{attribute 'linkalways'} 
{attribute 'no_explicit_call' := 'This FB is a CLASS and must be accessed using methods or properties'}
{attribute 'enable_dynamic_creation'}
FUNCTION_BLOCK _ETcVnRTrees EXTENDS EnumDatatypeBase
VAR
	localData : ETcVnRTrees;
	activeData : REFERENCE TO ETcVnRTrees;
	enumBaseDatatype : _UDINT(localData);
END_VAR

METHOD PRIVATE AddLocalEnumeration
VAR_INPUT
	Enumeration : T_MAXSTRING;
	Value : ETcVnRTrees;
END_VAR
AddEnumeration(Enumeration, Value);
END_METHOD

PROPERTY PUBLIC Address : PVOID
GET
Address := ADR(activeData);
END_GET
END_PROPERTY

METHOD PUBLIC ClearReference
VAR_INPUT
END_VAR
activeData REF= localData;
SetBaseDatatypeReference();
END_METHOD

METHOD PUBLIC Clone : I_Datatype
VAR
    pClone : POINTER TO _ETcVnRTrees;
END_VAR
pClone := __NEW(_ETcVnRTrees(InitialValue := Value));
Clone := pClone^;
END_METHOD

METHOD FB_init : BOOL
VAR_INPUT
	bInitRetains : BOOL; // if TRUE, the retain variables are initialized (warm start / cold start)
	bInCopyCode : BOOL;  // if TRUE, the instance afterwards gets moved into the copy code (online change)
	InitialValue : ETcVnRTrees;
END_VAR
localData := InitialValue;
AddBaseDatatype(enumBaseDatatype);
ClearReference();

AddLocalEnumeration('TCVN_RT_CLASSIFIER', ETcVnRTrees.TCVN_RT_CLASSIFIER);
AddLocalEnumeration('TCVN_RT_REGRESSOR', ETcVnRTrees.TCVN_RT_REGRESSOR);
END_METHOD

PROPERTY PUBLIC Identifier : T_MAXSTRING
GET
Identifier := 'ETcVnRTrees';
END_GET
END_PROPERTY

METHOD IsEnumeratorValueEqual : BOOL
VAR_INPUT
	Enumerator : I_KeyValueForwardEnumerator;
END_VAR
VAR
	storedValue : ETcVnRTrees;
END_VAR
IF NOT Enumerator.TryGet(storedValue) THEN
	RETURN;
END_IF

IsEnumeratorValueEqual := storedValue = activeData;
END_METHOD

METHOD PUBLIC MakeReferenceTo
VAR_INPUT
	ReferenceTarget : REFERENCE TO ETcVnRTrees;
END_VAR
activeData REF= ReferenceTarget;
SetBaseDatatypeReference();
END_METHOD

METHOD PROTECTED SetBaseDatatypeReference
VAR_INPUT
END_VAR
enumBaseDatatype.MakeReferenceTo(activeData);
END_METHOD

PROPERTY PUBLIC Size : UDINT
GET
Size := SIZEOF(activeData);
END_GET
END_PROPERTY

METHOD TryMakeReferenceTo : BOOL
VAR_INPUT
	Target : I_Datatype;
END_VAR
VAR
	targetAsEnum : I_EnumDatatype;
	pTargetData : POINTER TO ETcVnRTrees;
END_VAR
IF NOT Target.TryResolveAsEnumDatatype(targetAsEnum) THEN
	RETURN;
END_IF

IF targetAsEnum.Identifier <> Identifier THEN
	RETURN;
END_IF

pTargetData := Target.Address;
activeData REF= pTargetData^;
SetBaseDatatypeReference();
TryMakeReferenceTo := TRUE;
END_METHOD

PROPERTY PUBLIC Value : ETcVnRTrees
GET
Value := activeData;
END_GET
SET
activeData := Value;
END_SET
END_PROPERTY

END_FUNCTION_BLOCK

(* stored: Version 1.1.0.1, ProductVersion 3.1.4024.12
   POU _ETcVnRTrees: Id {5121f43b-3ca2-4baf-bd5c-a2722b22dd51}, SpecialFunc None
   Folder Constructor: Id {2dcca765-5c1c-4e5d-8a56-08c78f1e00a4}
   Folder Private: Id {82459e84-156f-4780-8edb-40ba5a89ab1f}
   Folder Protected: Id {f1614cfd-2cbd-46a2-8779-fde5d5b4e889}
   Method AddLocalEnumeration: Id {f0e52ad1-1d34-4ede-a2cc-4e0a7a0d8418}
   Property Address: Id {9145cbc1-482e-46a9-827a-d012f0b537b2}
   Get Get: Id {a8be51ba-dc92-49a6-8362-87afc485e47c}
   Method ClearReference: Id {c0f97e4c-1bce-44dd-8907-1b9faa6307e1}
   Method Clone: Id {90d92231-6005-4cd3-8df1-f7a9a1dbe83f}
   Method FB_init: Id {6950f6ed-de11-408d-a40e-14c5c9879686}
   Property Identifier: Id {50df2631-3018-4b3a-af29-e7d074cc9a69}
   Get Get: Id {3007bfd1-fbc2-48c1-a2f5-7da496783e77}
   Method IsEnumeratorValueEqual: Id {f60bf6ea-fc78-4cb1-8f02-a5cbbd486537}
   Method MakeReferenceTo: Id {9ad1ef7e-4852-4937-b4e9-c32b74d5627f}
   Method SetBaseDatatypeReference: Id {834773ac-0ab1-493d-8ea5-c9b79d884c41}
   Property Size: Id {7e10fbde-d8fe-4c6f-8e66-1153a986247c}
   Get Get: Id {70c8378b-ce85-4599-9a97-56ebe4935fe2}
   Method TryMakeReferenceTo: Id {18390fd8-b625-4058-b41e-89b9468d9c36}
   Property Value: Id {b77d6ad1-93b0-4872-b4a4-622c8836207a}
   Get Get: Id {a8af7cb5-5162-4a57-b6bb-0c60dfa5b637}
   Set Set: Id {9f836f23-0a4d-4a87-b164-3185e07c49b6} *)
